// Implicitly generated code : DO NOT EDIT
FUNCTION CheckBounds : DINT
VAR_INPUT
	index, lower, upper: DINT;
END_VAR

// Implicitly generated code : Only an Implementation suggestion
IF  index < lower THEN
	CheckBounds := lower;
	GVL_Checks.dCheckBounds := GVL_Checks.dCheckBounds + 1;
	ADSLOGSTR(4,'Checks critical error - index out of range','');
ELSIF  index > upper THEN
	CheckBounds := upper;
	GVL_Checks.dCheckBounds := GVL_Checks.dCheckBounds + 1;
	ADSLOGSTR(4,'Checks critical error - index out of range','');
ELSE  
	CheckBounds := index;
END_IF

END_FUNCTION

(* stored: Version 1.1.0.1, ProductVersion 3.1.4022.18
   POU CheckBounds: Id {a2917252-a5bd-462b-898a-66626a9a5ae1}, SpecialFunc CheckBounds *)
